{attribute 'GeneratedUsingTerminal: EJ9576-0000-0019'}
{attribute addProperty BoxType "EJ9576-0000-0019"}
{attribute addProperty Id "EtcSlaveTerminalBaseBCT_InputsAT %I*BCT_Inputs_4B98789517WcStateAT %I*WcState_9091E0EB2InfoDataAT %I*InfoData_32EB74EA10"}
{attribute addProperty CRC "2273633773"}
{attribute addProperty Size "29"}
TYPE EJ9576_8784E5ED EXTENDS EtcSlaveTerminalBase :
STRUCT
	{attribute addProperty Name "BCT_Inputs"}
	BCT_Inputs : BCT_Inputs_4B987895;
	{attribute addProperty Name "WcState"}
	WcState : WcState_9091E0EB;
	{attribute addProperty Name "InfoData"}
	InfoData : InfoData_32EB74EA;
END_STRUCT
END_TYPE

(* stored: Version 1.2.0.0, ProductVersion 3.1.4024.9
   DUT EJ9576_8784E5ED: Id {8c561cb4-4b3d-40fd-9525-23fc7eb65827} *)
